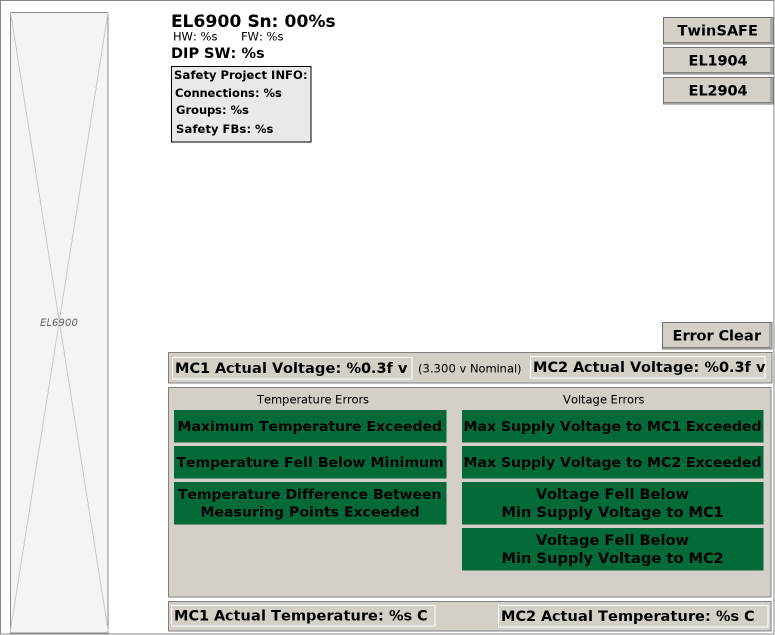
VISUALIZATION EL6900_Specific_Diagnostics  // 775x635
    Button (663,17 110x27), "TwinSAFE"
        OnMouseClick: change screen: TwinSAFE
    Button (663,47 110x27), "EL1904"
        OnMouseClick: change screen: EL1904_Specific_Diagnostics
    Button (663,77 110x27), "EL2904"
        OnMouseClick: change screen: EL2904_Specific_Diagnostics
    Image (10,12 98x621), image: EL6900
    Rectangle (168,10 275x22), "EL6900 Sn: 00%s", text variable: g_dwHMI_EL6900Sn
    Rectangle (170,28 65x17), "HW: %s", text variable: g_sHMI_EL6900_HWvers
    Rectangle (238,28 65x17), "FW: %s", text variable: g_sHMI_EL6900_FWvers
    Rectangle (168,42 164x22), "DIP SW: %s", text variable: g_wHMI_EL6900DSw
    Group (171,64 140x78)
        Rectangle (0,2 140x76)
        Rectangle (1,17 135x24), "Connections: %s", text variable: g_bHMI_EL6900_NoOfConnections
        Label (0,0 135x22), "Safety Project INFO:"
        Rectangle (2,34 135x24), "Groups: %s", text variable: g_bHMI_EL6900_NoOfSafetyGrps
        Rectangle (2,53 135x24), "Safety FBs: %s", text variable: g_bHMI_EL6900_NoOfSafetyFBs
    Button (662,322 110x27), "Error Clear"
        OnMouseUp: execute { g_xHMI_EL6900_ErrClearPB := FALSE ; }
        OnMouseDown: execute { g_xHMI_EL6900_ErrClearPB := TRUE ; }
    Group (168,352 604x31)
        Rectangle (0,0 604x31)
        Label (243,9 118x15), "(3.300 v Nominal)"
        Rectangle (4,5 240x22), "MC1 Actual Voltage: %0.3f v", text variable: g_wHMI_EL6900PriMC_Volts
        Rectangle (362,4 235x22), "MC2 Actual Voltage: %0.3f v", text variable: g_wHMI_EL6900SecMC_Volts
    Group (168,601 603x30)
        Rectangle (0,0 603x30)
        Rectangle (3,4 264x21), "MC1 Actual Temperature: %s C", text variable: g_wHMI_EL6900PriMCTemp
        Rectangle (330,4 270x22), "MC2 Actual Temperature: %s C", text variable: g_wHMI_EL6900SecMCTemp
    Group (168,387 603x210)
        Rectangle (0,0 603x210)
        Label (80,0 130x25), "Temperature Errors"
        Rectangle (6,23 272x32), "Maximum Temperature Exceeded", colour toggle: g_xHMI_EL6900_MaxTemp
        Label (371,0 130x25), "Voltage Errors"
        Rectangle (6,59 272x32), "Temperature Fell Below Minimum", colour toggle: g_xHMI_EL6900_MinTemp
        Rectangle (6,95 272x42), "Temperature Difference Between Measuring Points Exceeded", colour toggle: g_xHMI_EL6900_TempDiffExceeded
        Rectangle (294,23 301x32), "Max Supply Voltage to MC1 Exceeded", colour toggle: g_xHMI_EL6900_MaxVccMC1
        Rectangle (294,59 301x32), "Max Supply Voltage to MC2 Exceeded", colour toggle: g_xHMI_EL6900_MaxVccMC2
        Rectangle (294,95 301x42), "Voltage Fell Below Min Supply Voltage to MC1", colour toggle: g_xHMI_EL6900_MinVccMC1
        Rectangle (294,141 301x42), "Voltage Fell Below Min Supply Voltage to MC2", colour toggle: g_xHMI_EL6900_MinVccMC2
END_VISUALIZATION

(* stored: Version 1.1.0.1, ProductVersion 3.1.0.18
   Visu EL6900_Specific_Diagnostics: Id {afbb687b-b013-47d9-9512-f6b712c2fba3} *)
